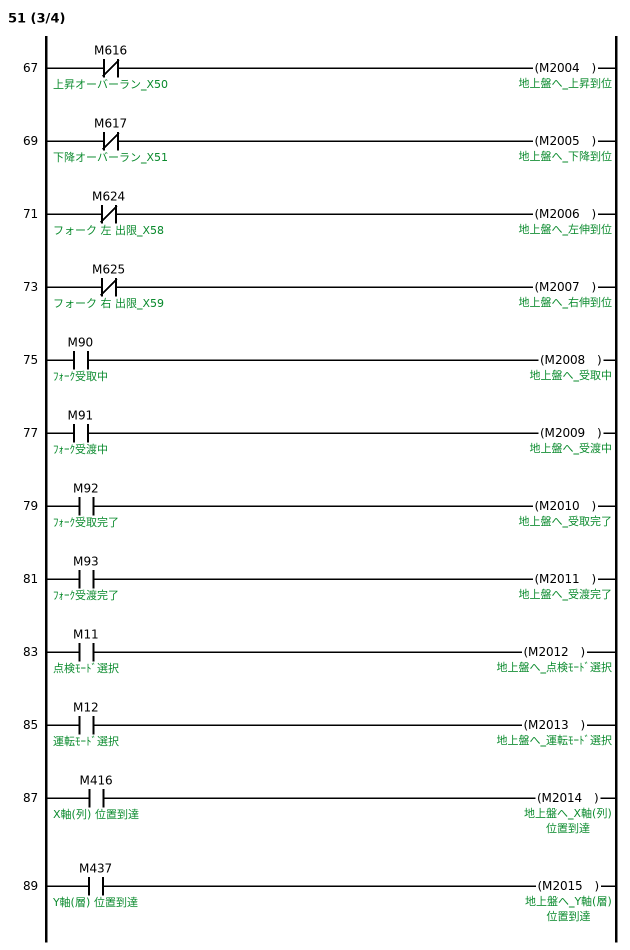
67    LDI     M616  ; 上昇オーバーラン_X50
      OUT     M2004  ; 地上盤へ_上昇到位
69    LDI     M617  ; 下降オーバーラン_X51
      OUT     M2005  ; 地上盤へ_下降到位
71    LDI     M624  ; フォーク 左 出限_X58
      OUT     M2006  ; 地上盤へ_左伸到位
73    LDI     M625  ; フォーク 右 出限_X59
      OUT     M2007  ; 地上盤へ_右伸到位
75    LD      M90  ; ﾌｫｰｸ受取中
      OUT     M2008  ; 地上盤へ_受取中
77    LD      M91  ; ﾌｫｰｸ受渡中
      OUT     M2009  ; 地上盤へ_受渡中
79    LD      M92  ; ﾌｫｰｸ受取完了
      OUT     M2010  ; 地上盤へ_受取完了
81    LD      M93  ; ﾌｫｰｸ受渡完了
      OUT     M2011  ; 地上盤へ_受渡完了
83    LD      M11  ; 点検ﾓｰﾄﾞ選択
      OUT     M2012  ; 地上盤へ_点検ﾓｰﾄﾞ選択
85    LD      M12  ; 運転ﾓｰﾄﾞ選択
      OUT     M2013  ; 地上盤へ_運転ﾓｰﾄﾞ選択
87    LD      M416  ; X軸(列) 位置到達
      OUT     M2014  ; 地上盤へ_X軸(列) 位置到達
89    LD      M437  ; Y軸(層) 位置到達
      OUT     M2015  ; 地上盤へ_Y軸(層) 位置到達
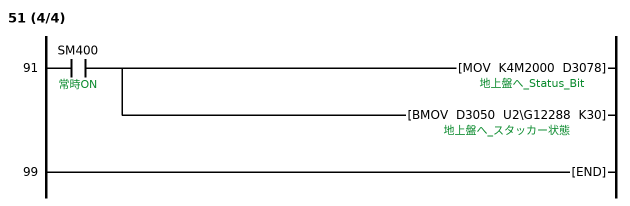
91    LD      SM400  ; 常時ON
      MOV     K4M2000 D3078  ; 地上盤へ_Status_Bit
      BMOV    D3050 U2\G12288 K30
99    END
END_PROGRAM

PROGRAM 52  // Ether 出力 SEW INV
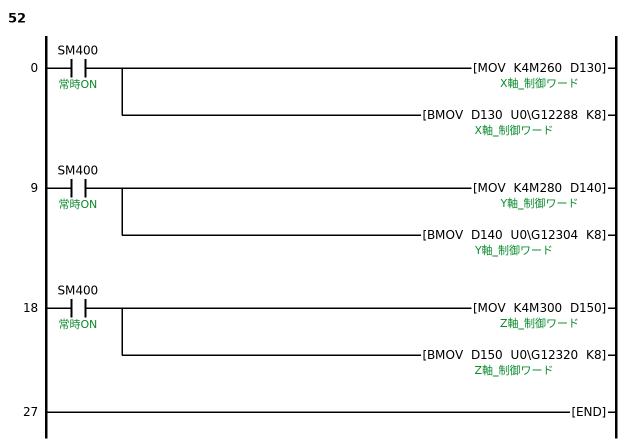
0     LD      SM400  ; 常時ON
      MOV     K4M260 D130  ; X軸_Enable非常停止 / X軸_制御ワード
      BMOV    D130 U0\G12288 K8
9     LD      SM400  ; 常時ON
      MOV     K4M280 D140  ; Y軸_Enable非常停止 / Y軸_制御ワード
      BMOV    D140 U0\G12304 K8
18    LD      SM400  ; 常時ON
      MOV     K4M300 D150  ; Z軸_Enable非常停止 / Z軸_制御ワード
      BMOV    D150 U0\G12320 K8
27    END
END_PROGRAM

PROGRAM 01  // IO入力
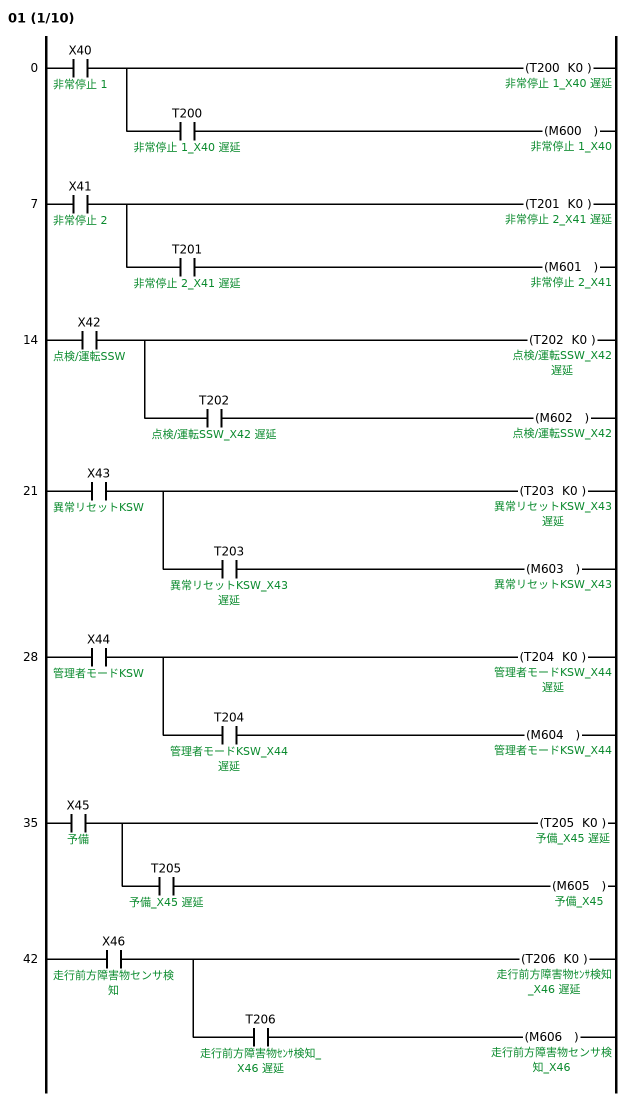
0     LD      X40  ; 非常停止 1
      OUT     T200 K0  ; 非常停止 1_X40 遅延
      AND     T200  ; 非常停止 1_X40 遅延
      OUT     M600  ; 非常停止 1_X40
7     LD      X41  ; 非常停止 2
      OUT     T201 K0  ; 非常停止 2_X41 遅延
      AND     T201  ; 非常停止 2_X41 遅延
      OUT     M601  ; 非常停止 2_X41
14    LD      X42  ; 点検/運転SSW
      OUT     T202 K0  ; 点検/運転SSW_X42 遅延
      AND     T202  ; 点検/運転SSW_X42 遅延
      OUT     M602  ; 点検/運転SSW_X42
21    LD      X43  ; 異常リセットKSW
      OUT     T203 K0  ; 異常リセットKSW_X43 遅延
      AND     T203  ; 異常リセットKSW_X43 遅延
      OUT     M603  ; 異常リセットKSW_X43
28    LD      X44  ; 管理者モードKSW
      OUT     T204 K0  ; 管理者モードKSW_X44 遅延
      AND     T204  ; 管理者モードKSW_X44 遅延
      OUT     M604  ; 管理者モードKSW_X44
35    LD      X45  ; 予備
      OUT     T205 K0  ; 予備_X45 遅延
      AND     T205  ; 予備_X45 遅延
      OUT     M605  ; 予備_X45
42    LD      X46  ; 走行前方障害物センサ検知
      OUT     T206 K0  ; 走行前方障害物ｾﾝｻ検知_X46 遅延
      AND     T206  ; 走行前方障害物ｾﾝｻ検知_X46 遅延
      OUT     M606  ; 走行前方障害物センサ検知_X46
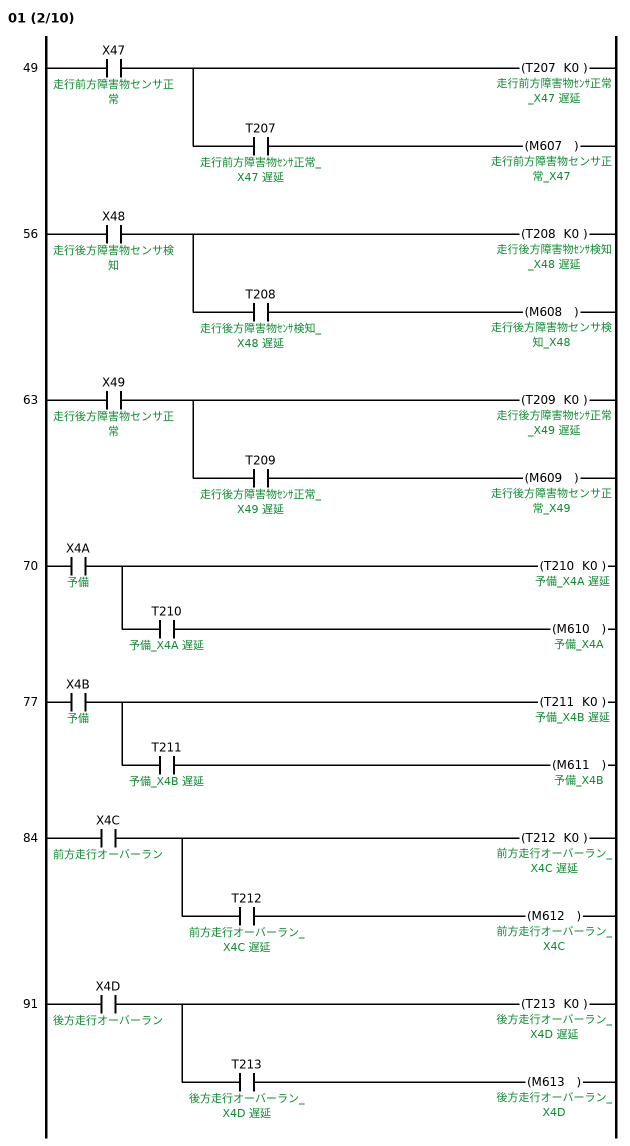
49    LD      X47  ; 走行前方障害物センサ正常
      OUT     T207 K0  ; 走行前方障害物ｾﾝｻ正常_X47 遅延
      AND     T207  ; 走行前方障害物ｾﾝｻ正常_X47 遅延
      OUT     M607  ; 走行前方障害物センサ正常_X47
56    LD      X48  ; 走行後方障害物センサ検知
      OUT     T208 K0  ; 走行後方障害物ｾﾝｻ検知_X48 遅延
      AND     T208  ; 走行後方障害物ｾﾝｻ検知_X48 遅延
      OUT     M608  ; 走行後方障害物センサ検知_X48
63    LD      X49  ; 走行後方障害物センサ正常
      OUT     T209 K0  ; 走行後方障害物ｾﾝｻ正常_X49 遅延
      AND     T209  ; 走行後方障害物ｾﾝｻ正常_X49 遅延
      OUT     M609  ; 走行後方障害物センサ正常_X49
70    LD      X4A  ; 予備
      OUT     T210 K0  ; 予備_X4A 遅延
      AND     T210  ; 予備_X4A 遅延
      OUT     M610  ; 予備_X4A
77    LD      X4B  ; 予備
      OUT     T211 K0  ; 予備_X4B 遅延
      AND     T211  ; 予備_X4B 遅延
      OUT     M611  ; 予備_X4B
84    LD      X4C  ; 前方走行オーバーラン
      OUT     T212 K0  ; 前方走行オーバーラン_X4C 遅延
      AND     T212  ; 前方走行オーバーラン_X4C 遅延
      OUT     M612  ; 前方走行オーバーラン_X4C
91    LD      X4D  ; 後方走行オーバーラン
      OUT     T213 K0  ; 後方走行オーバーラン_X4D 遅延
      AND     T213  ; 後方走行オーバーラン_X4D 遅延
      OUT     M613  ; 後方走行オーバーラン_X4D
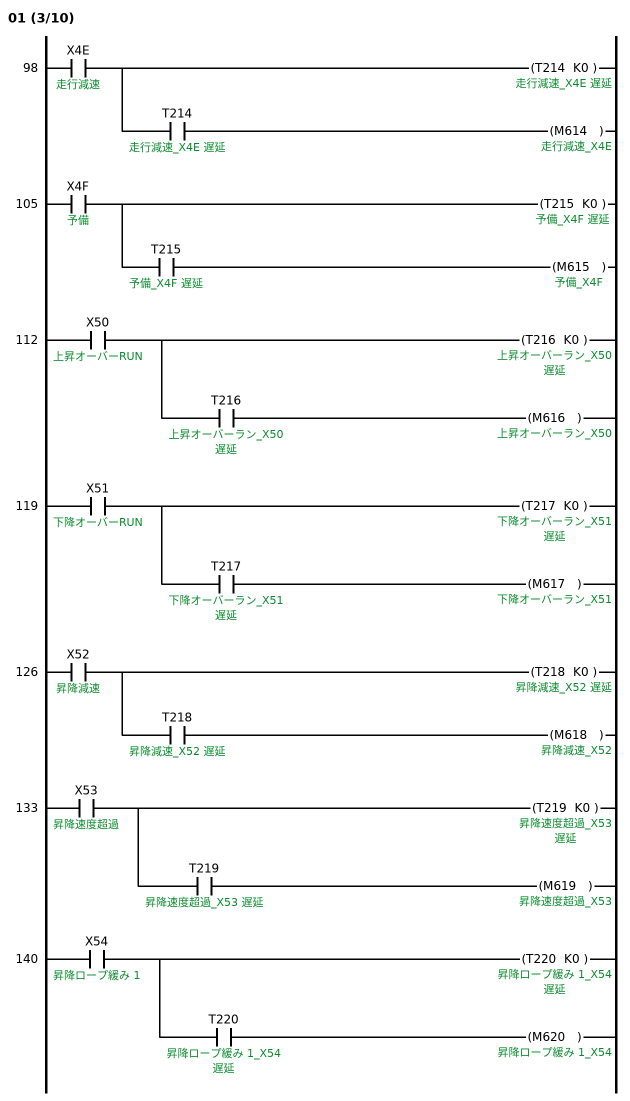
98    LD      X4E  ; 走行減速
      OUT     T214 K0  ; 走行減速_X4E 遅延
      AND     T214  ; 走行減速_X4E 遅延
      OUT     M614  ; 走行減速_X4E
105   LD      X4F  ; 予備
      OUT     T215 K0  ; 予備_X4F 遅延
      AND     T215  ; 予備_X4F 遅延
      OUT     M615  ; 予備_X4F
112   LD      X50  ; 上昇オーバーRUN
      OUT     T216 K0  ; 上昇オーバーラン_X50 遅延
      AND     T216  ; 上昇オーバーラン_X50 遅延
      OUT     M616  ; 上昇オーバーラン_X50
119   LD      X51  ; 下降オーバーRUN
      OUT     T217 K0  ; 下降オーバーラン_X51 遅延
      AND     T217  ; 下降オーバーラン_X51 遅延
      OUT     M617  ; 下降オーバーラン_X51
126   LD      X52  ; 昇降減速
      OUT     T218 K0  ; 昇降減速_X52 遅延
      AND     T218  ; 昇降減速_X52 遅延
      OUT     M618  ; 昇降減速_X52
133   LD      X53  ; 昇降速度超過
      OUT     T219 K0  ; 昇降速度超過_X53 遅延
      AND     T219  ; 昇降速度超過_X53 遅延
      OUT     M619  ; 昇降速度超過_X53
140   LD      X54  ; 昇降ロープ緩み 1
      OUT     T220 K0  ; 昇降ロープ緩み 1_X54 遅延
      AND     T220  ; 昇降ロープ緩み 1_X54 遅延
      OUT     M620  ; 昇降ロープ緩み 1_X54
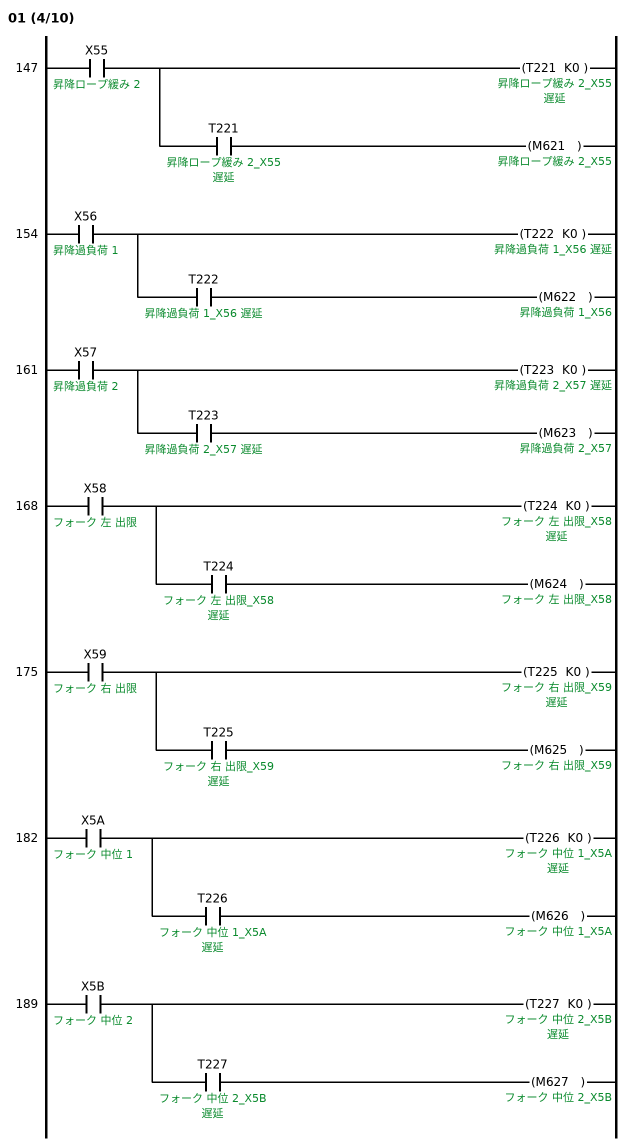
147   LD      X55  ; 昇降ロープ緩み 2
      OUT     T221 K0  ; 昇降ロープ緩み 2_X55 遅延
      AND     T221  ; 昇降ロープ緩み 2_X55 遅延
      OUT     M621  ; 昇降ロープ緩み 2_X55
154   LD      X56  ; 昇降過負荷 1
      OUT     T222 K0  ; 昇降過負荷 1_X56 遅延
      AND     T222  ; 昇降過負荷 1_X56 遅延
      OUT     M622  ; 昇降過負荷 1_X56
161   LD      X57  ; 昇降過負荷 2
      OUT     T223 K0  ; 昇降過負荷 2_X57 遅延
      AND     T223  ; 昇降過負荷 2_X57 遅延
      OUT     M623  ; 昇降過負荷 2_X57
168   LD      X58  ; フォーク 左 出限
      OUT     T224 K0  ; フォーク 左 出限_X58 遅延
      AND     T224  ; フォーク 左 出限_X58 遅延
      OUT     M624  ; フォーク 左 出限_X58
175   LD      X59  ; フォーク 右 出限
      OUT     T225 K0  ; フォーク 右 出限_X59 遅延
      AND     T225  ; フォーク 右 出限_X59 遅延
      OUT     M625  ; フォーク 右 出限_X59
182   LD      X5A  ; フォーク 中位 1
      OUT     T226 K0  ; フォーク 中位 1_X5A 遅延
      AND     T226  ; フォーク 中位 1_X5A 遅延
      OUT     M626  ; フォーク 中位 1_X5A
189   LD      X5B  ; フォーク 中位 2
      OUT     T227 K0  ; フォーク 中位 2_X5B 遅延
      AND     T227  ; フォーク 中位 2_X5B 遅延
      OUT     M627  ; フォーク 中位 2_X5B
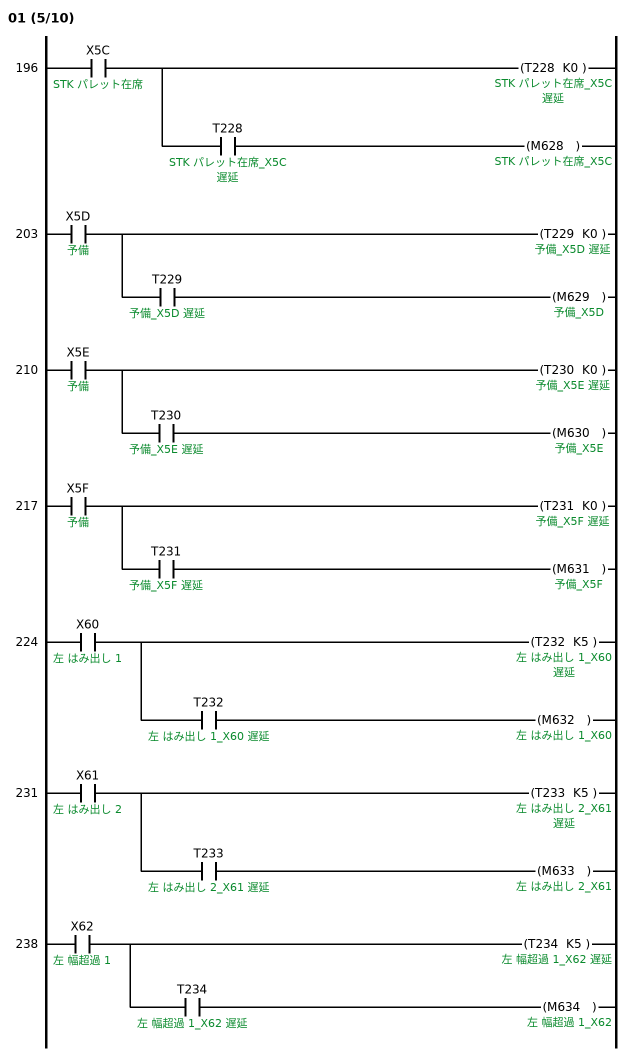
196   LD      X5C  ; STK パレット在席
      OUT     T228 K0  ; STK パレット在席_X5C 遅延
      AND     T228  ; STK パレット在席_X5C 遅延
      OUT     M628  ; STK パレット在席_X5C
203   LD      X5D  ; 予備
      OUT     T229 K0  ; 予備_X5D 遅延
      AND     T229  ; 予備_X5D 遅延
      OUT     M629  ; 予備_X5D
210   LD      X5E  ; 予備
      OUT     T230 K0  ; 予備_X5E 遅延
      AND     T230  ; 予備_X5E 遅延
      OUT     M630  ; 予備_X5E
217   LD      X5F  ; 予備
      OUT     T231 K0  ; 予備_X5F 遅延
      AND     T231  ; 予備_X5F 遅延
      OUT     M631  ; 予備_X5F
224   LD      X60  ; 左 はみ出し 1
      OUT     T232 K5  ; 左 はみ出し 1_X60 遅延
      AND     T232  ; 左 はみ出し 1_X60 遅延
      OUT     M632  ; 左 はみ出し 1_X60
231   LD      X61  ; 左 はみ出し 2
      OUT     T233 K5  ; 左 はみ出し 2_X61 遅延
      AND     T233  ; 左 はみ出し 2_X61 遅延
      OUT     M633  ; 左 はみ出し 2_X61
238   LD      X62  ; 左 幅超過 1
      OUT     T234 K5  ; 左 幅超過 1_X62 遅延
      AND     T234  ; 左 幅超過 1_X62 遅延
      OUT     M634  ; 左 幅超過 1_X62
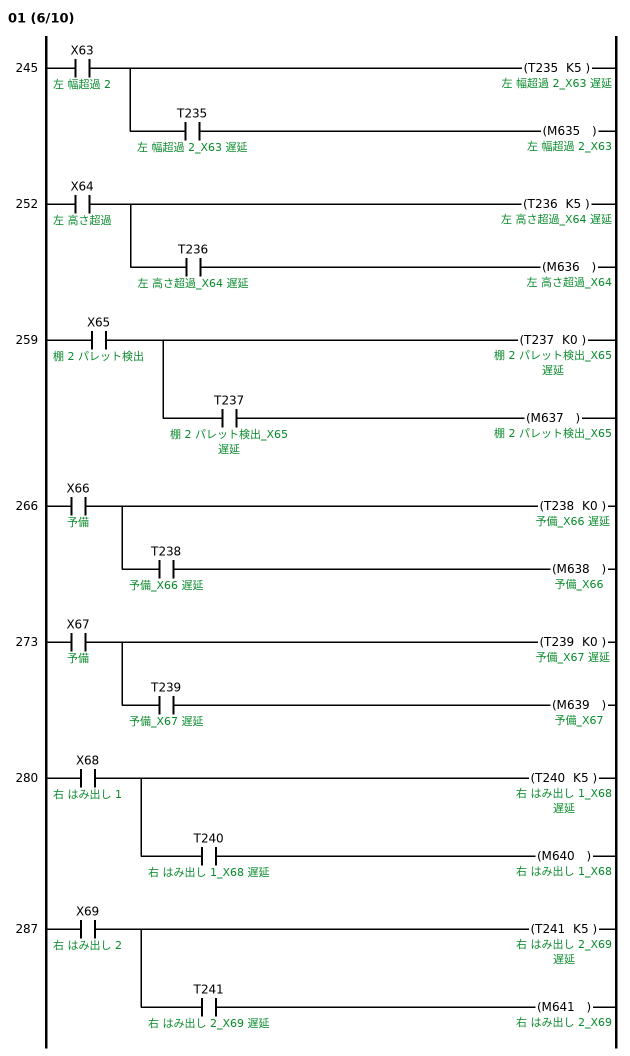
245   LD      X63  ; 左 幅超過 2
      OUT     T235 K5  ; 左 幅超過 2_X63 遅延
      AND     T235  ; 左 幅超過 2_X63 遅延
      OUT     M635  ; 左 幅超過 2_X63
252   LD      X64  ; 左 高さ超過
      OUT     T236 K5  ; 左 高さ超過_X64 遅延
      AND     T236  ; 左 高さ超過_X64 遅延
      OUT     M636  ; 左 高さ超過_X64
259   LD      X65  ; 棚 2 パレット検出
      OUT     T237 K0  ; 棚 2 パレット検出_X65 遅延
      AND     T237  ; 棚 2 パレット検出_X65 遅延
      OUT     M637  ; 棚 2 パレット検出_X65
266   LD      X66  ; 予備
      OUT     T238 K0  ; 予備_X66 遅延
      AND     T238  ; 予備_X66 遅延
      OUT     M638  ; 予備_X66
273   LD      X67  ; 予備
      OUT     T239 K0  ; 予備_X67 遅延
      AND     T239  ; 予備_X67 遅延
      OUT     M639  ; 予備_X67
280   LD      X68  ; 右 はみ出し 1
      OUT     T240 K5  ; 右 はみ出し 1_X68 遅延
      AND     T240  ; 右 はみ出し 1_X68 遅延
      OUT     M640  ; 右 はみ出し 1_X68
287   LD      X69  ; 右 はみ出し 2
      OUT     T241 K5  ; 右 はみ出し 2_X69 遅延
      AND     T241  ; 右 はみ出し 2_X69 遅延
      OUT     M641  ; 右 はみ出し 2_X69
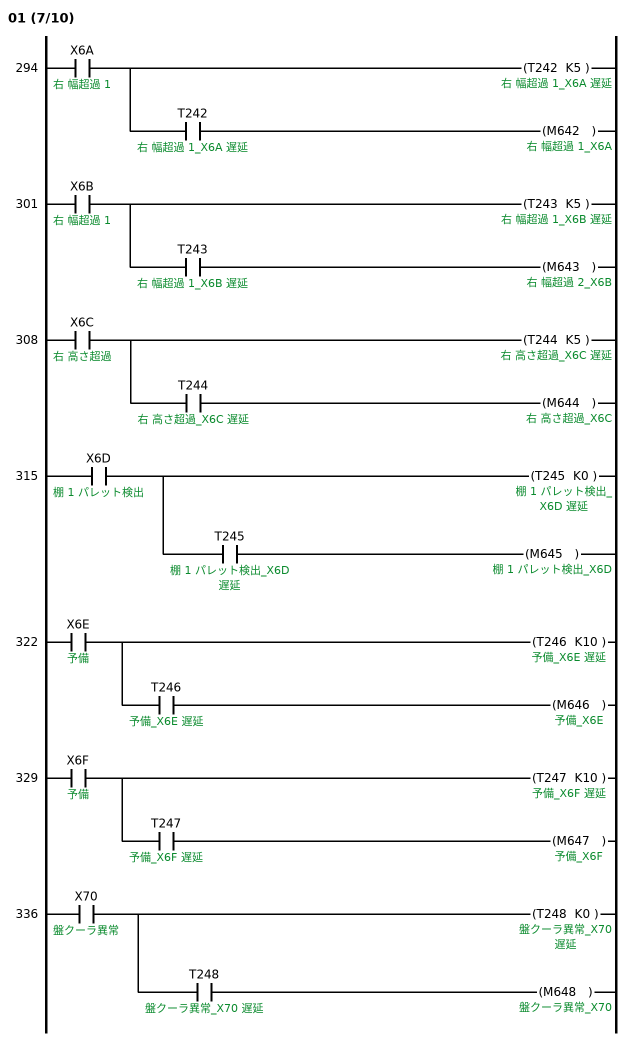
294   LD      X6A  ; 右 幅超過 1
      OUT     T242 K5  ; 右 幅超過 1_X6A 遅延
      AND     T242  ; 右 幅超過 1_X6A 遅延
      OUT     M642  ; 右 幅超過 1_X6A
301   LD      X6B  ; 右 幅超過 1
      OUT     T243 K5  ; 右 幅超過 1_X6B 遅延
      AND     T243  ; 右 幅超過 1_X6B 遅延
      OUT     M643  ; 右 幅超過 2_X6B
308   LD      X6C  ; 右 高さ超過
      OUT     T244 K5  ; 右 高さ超過_X6C 遅延
      AND     T244  ; 右 高さ超過_X6C 遅延
      OUT     M644  ; 右 高さ超過_X6C
315   LD      X6D  ; 棚 1 パレット検出
      OUT     T245 K0  ; 棚 1 パレット検出_X6D 遅延
      AND     T245  ; 棚 1 パレット検出_X6D 遅延
      OUT     M645  ; 棚 1 パレット検出_X6D
322   LD      X6E  ; 予備
      OUT     T246 K10  ; 予備_X6E 遅延
      AND     T246  ; 予備_X6E 遅延
      OUT     M646  ; 予備_X6E
329   LD      X6F  ; 予備
      OUT     T247 K10  ; 予備_X6F 遅延
      AND     T247  ; 予備_X6F 遅延
      OUT     M647  ; 予備_X6F
336   LD      X70  ; 盤クーラ異常
      OUT     T248 K0  ; 盤クーラ異常_X70 遅延
      AND     T248  ; 盤クーラ異常_X70 遅延
      OUT     M648  ; 盤クーラ異常_X70
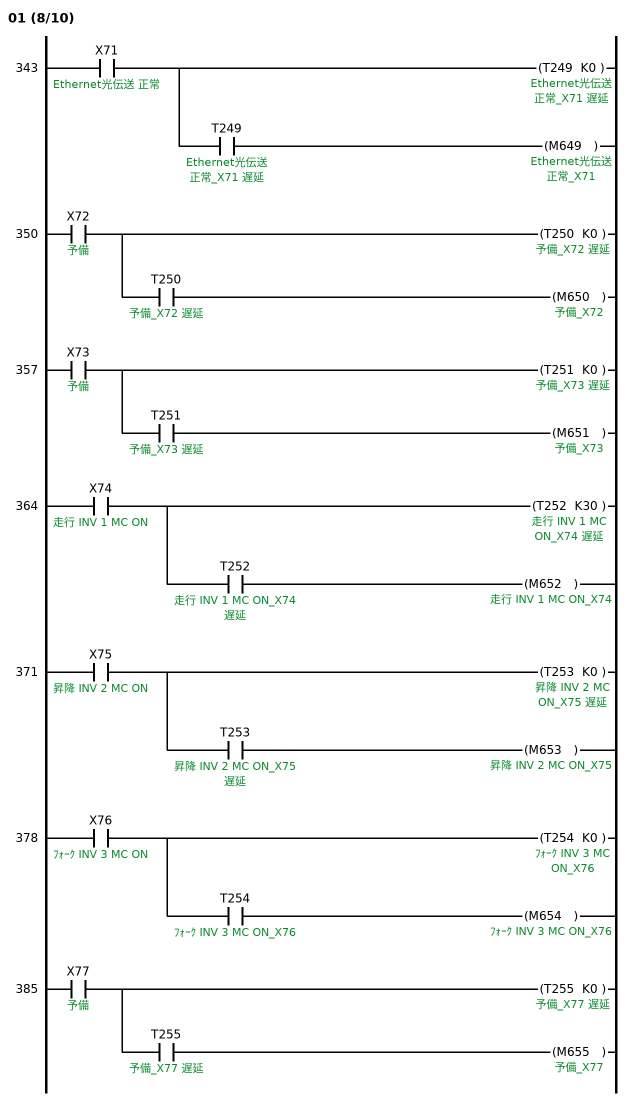
343   LD      X71  ; Ethernet光伝送 正常
      OUT     T249 K0  ; Ethernet光伝送 正常_X71 遅延
      AND     T249  ; Ethernet光伝送 正常_X71 遅延
      OUT     M649  ; Ethernet光伝送 正常_X71
350   LD      X72  ; 予備
      OUT     T250 K0  ; 予備_X72 遅延
      AND     T250  ; 予備_X72 遅延
      OUT     M650  ; 予備_X72
357   LD      X73  ; 予備
      OUT     T251 K0  ; 予備_X73 遅延
      AND     T251  ; 予備_X73 遅延
      OUT     M651  ; 予備_X73
364   LD      X74  ; 走行 INV 1 MC ON
      OUT     T252 K30  ; 走行 INV 1 MC ON_X74 遅延
      AND     T252  ; 走行 INV 1 MC ON_X74 遅延
      OUT     M652  ; 走行 INV 1 MC ON_X74
371   LD      X75  ; 昇降 INV 2 MC ON
      OUT     T253 K0  ; 昇降 INV 2 MC ON_X75 遅延
      AND     T253  ; 昇降 INV 2 MC ON_X75 遅延
      OUT     M653  ; 昇降 INV 2 MC ON_X75
378   LD      X76  ; ﾌｫｰｸ INV 3 MC ON
      OUT     T254 K0  ; ﾌｫｰｸ INV 3 MC ON_X76
      AND     T254  ; ﾌｫｰｸ INV 3 MC ON_X76
      OUT     M654  ; ﾌｫｰｸ INV 3 MC ON_X76
385   LD      X77  ; 予備
      OUT     T255 K0  ; 予備_X77 遅延
      AND     T255  ; 予備_X77 遅延
      OUT     M655  ; 予備_X77
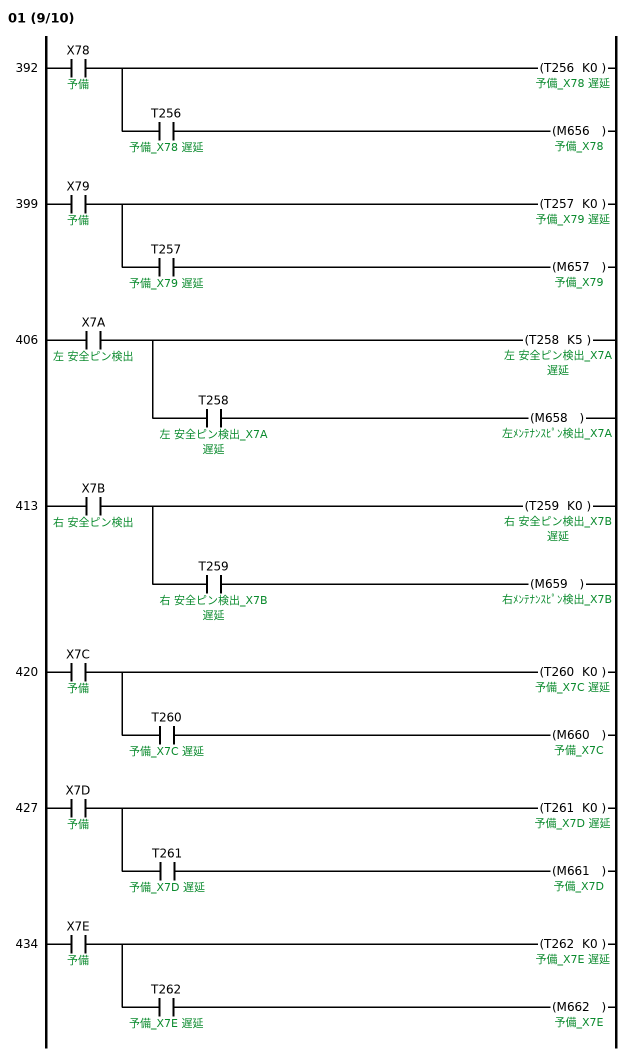
392   LD      X78  ; 予備
      OUT     T256 K0  ; 予備_X78 遅延
      AND     T256  ; 予備_X78 遅延
      OUT     M656  ; 予備_X78
399   LD      X79  ; 予備
      OUT     T257 K0  ; 予備_X79 遅延
      AND     T257  ; 予備_X79 遅延
      OUT     M657  ; 予備_X79
406   LD      X7A  ; 左 安全ピン検出
      OUT     T258 K5  ; 左 安全ピン検出_X7A 遅延
      AND     T258  ; 左 安全ピン検出_X7A 遅延
      OUT     M658  ; 左ﾒﾝﾃﾅﾝｽﾋﾟﾝ検出_X7A
413   LD      X7B  ; 右 安全ピン検出
      OUT     T259 K0  ; 右 安全ピン検出_X7B 遅延
      AND     T259  ; 右 安全ピン検出_X7B 遅延
      OUT     M659  ; 右ﾒﾝﾃﾅﾝｽﾋﾟﾝ検出_X7B
420   LD      X7C  ; 予備
      OUT     T260 K0  ; 予備_X7C 遅延
      AND     T260  ; 予備_X7C 遅延
      OUT     M660  ; 予備_X7C
427   LD      X7D  ; 予備
      OUT     T261 K0  ; 予備_X7D 遅延
      AND     T261  ; 予備_X7D 遅延
      OUT     M661  ; 予備_X7D
434   LD      X7E  ; 予備
      OUT     T262 K0  ; 予備_X7E 遅延
      AND     T262  ; 予備_X7E 遅延
      OUT     M662  ; 予備_X7E
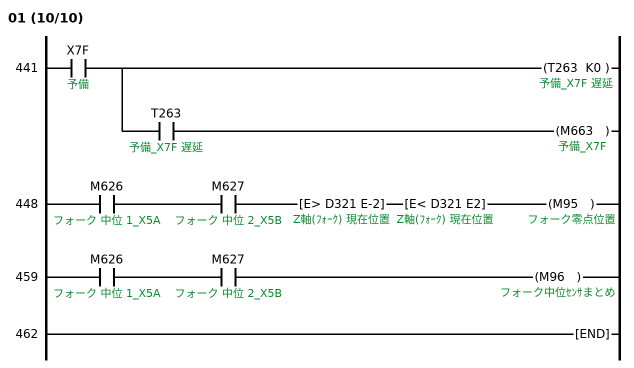
441   LD      X7F  ; 予備
      OUT     T263 K0  ; 予備_X7F 遅延
      AND     T263  ; 予備_X7F 遅延
      OUT     M663  ; 予備_X7F
448   LD      M626  ; フォーク 中位 1_X5A
      AND     M627  ; フォーク 中位 2_X5B
      ANDE>   D321 E-2  ; Z軸(ﾌｫｰｸ) 現在位置
      ANDE<   D321 E2  ; Z軸(ﾌｫｰｸ) 現在位置
      OUT     M95  ; フォーク零点位置
459   LD      M626  ; フォーク 中位 1_X5A
      AND     M627  ; フォーク 中位 2_X5B
      OUT     M96  ; フォーク中位ｾﾝｻまとめ
462   END
END_PROGRAM

// device comments not shown above
D3270  ; ﾌｫｰｸ座標  [1]
M0  ; 電源ON後遅延
M70  ; 待機 補助
M74  ; 受取位置へ 補助
M79  ; 受渡点へ 補助
M147  ; Z軸ON 位置決め_自動_補助 6
M148  ; Z軸ON 位置決め_自動_補助 7
M149  ; Z軸ON 位置決め_自動_補助 8
M201  ; X軸_STO非アクティブ
M202  ; X軸_出力段Enabled
M203  ; X軸_ブレーキオープン済み
M204  ; X軸_モーター回転
M206  ; X軸_新しい相対位置適用済み
M209  ; X軸_ワーニング
M210  ; X軸_ドライブ機構2 有効
M211  ; X軸_メッセージ実速度比較
M212  ; X軸_リミットスイッチ非アク
M213  ; X軸_予備
M214  ; X軸_待機運転有効
M215  ; X軸_HandshakeOut
M221  ; Y軸_STO非アクティブ
M222  ; Y軸_出力段已Enable
M223  ; Y軸_ブレーキオープン済み
M224  ; Y軸_モーター回転
M226  ; Y軸_新しい相対位置適用済み
M229  ; Y軸_ワーニング
M230  ; Y軸_ドライブ機構2 有効
M231  ; Y軸_メッセージ実速度比較
M232  ; Y軸_リミットスイッチ非アク
M233  ; Y軸_予備
M235  ; Y軸_HandshakeOut
M241  ; Z軸_STO非アクティブ
M242  ; Z軸_出力段已Enable
M243  ; Z軸_ブレーキオープン済み
M244  ; Z軸_モーター回転
M246  ; Z軸_新しい相対位置適用済み
M249  ; Z軸_ワーニング
M250  ; Z軸_ドライブ機構2 有効
M251  ; Z軸_メッセージ実速度比較
M252  ; Z軸_リミットスイッチ非アク
M253  ; Z軸_予備
M254  ; Z軸_待機運転有効
M255  ; Z軸_HandshakeOut
M262  ; X軸_予備1
M263  ; X軸_ブレーキ開放
M266  ; X軸_相対位置受信中
M269  ; X軸_予備2
M270  ; X軸_ドライブ機構2 有効
M271  ; X軸_予備3
M272  ; X軸_禁用リミットスイッ
M273  ; X軸_出力段ロック 有効
M274  ; X軸_待機運転有効
M275  ; X軸_HandshakeIn
M282  ; Y軸_予備1
M283  ; Y軸_ブレーキ開放
M286  ; Y軸_相対位置受信中
M289  ; Y軸_予備2
M291  ; Y軸_予備3
M292  ; Y軸_禁用リミットスイッ
M293  ; Y軸_出力段ロック 有効
M295  ; Y軸_HandshakeIn
M302  ; Z軸_予備1
M303  ; Z軸_ブレーキ開放
M306  ; Z軸_相対位置受信中
M309  ; Z軸_予備2
M310  ; Z軸_駆動機構作動
M311  ; Z軸_予備3
M312  ; Z軸_禁用リミットスイッ
M313  ; Z軸_出力段ロック 有効
M314  ; Z軸_待機運転有効
M315  ; Z軸_HandshakeIn
M400  ; X軸ON 位置決め0
M403  ; X軸ON 位置決め3
M404  ; X軸ON 位置決め4
M405  ; X軸ON 位置決め5
M406  ; X軸ON 位置決め6
M407  ; X軸ON 位置決め7
M408  ; X軸ON 位置決め8
M409  ; X軸ON 位置決め9
M410  ; X軸ON 位置決め10
M411  ; X軸ON 位置決め11
M412  ; X軸ON 位置決め12
M413  ; X軸ON 位置決め13
M414  ; X軸ON 位置決め14
M415  ; X軸ON 位置決め15
M421  ; Y軸ON 位置決め0
M424  ; Y軸ON 位置決め3
M425  ; Y軸ON 位置決め4
M426  ; Y軸ON 位置決め5
M427  ; Y軸ON 位置決め6
M428  ; Y軸ON 位置決め7
M429  ; Y軸ON 位置決め8
M430  ; Y軸ON 位置決め9
M431  ; Y軸ON 位置決め10
M432  ; Y軸ON 位置決め11
M433  ; Y軸ON 位置決め12
M434  ; Y軸ON 位置決め13
M435  ; Y軸ON 位置決め14
M436  ; Y軸ON 位置決め15
M442  ; Z軸ON 位置決め0
M445  ; Z軸ON 位置決め3
M446  ; Z軸ON 位置決め4
M447  ; Z軸ON 位置決め5
M448  ; Z軸ON 位置決め6
M449  ; Z軸ON 位置決め7
M450  ; Z軸ON 位置決め8
M451  ; Z軸ON 位置決め9
M452  ; Z軸ON 位置決め10
M453  ; Z軸ON 位置決め11
M454  ; Z軸ON 位置決め12
M455  ; Z軸ON 位置決め13
M456  ; Z軸ON 位置決め14
M457  ; Z軸ON 位置決め15
M921  ; 安全機器一時解除有効
M990  ; テスト用
M2514  ; 地上盤から_予備3
M2515  ; 地上盤から_予備4
M2516  ; 地上盤から_予備5
M2517  ; 地上盤から_予備6
M3196  ; フォーク右側超高アラーム
M3197  ; フォーク右超ワイドアラーム2
M3198  ; フォーク右超ワイドアラーム1
M3199  ; フォーク右側崩壊アラーム2
M3200  ; フォーク右側崩壊アラーム1
M3201  ; フォーク左側超高アラーム
M3202  ; フォーク左超ワイドアラーム2
M3203  ; フォーク左超ワイドアラーム1
M3204  ; フォーク左側崩壊アラーム2
M3205  ; フォーク左側崩壊アラーム1
M3206  ; 搬入可能
M3207  ; 搬出可能
M3230  ; DockTable1搬入可能2
M3231  ; DockTable2搬入可能2
M3232  ; DockTable1搬出可能1
M3233  ; DockTable2搬出可能1
D2  ; GOTｵｰﾊﾞﾗｯﾌﾟｳｨﾝﾄﾞｳ2
D3  ; GOTｵｰﾊﾞﾗｯﾌﾟｳｨﾝﾄﾞｳ3
D4  ; GOTｵｰﾊﾞﾗｯﾌﾟｳｨﾝﾄﾞｳ4
D5  ; GOTｵｰﾊﾞﾗｯﾌﾟｳｨﾝﾄﾞｳ5
D10  ; GOTｼｽﾃﾑ信号1-1
D11  ; GOTｼｽﾃﾑ信号2-1
D12  ; GOT表示中画面番号
D13  ; 表示中ｳｨﾝﾄﾞｳ画面1番号
D14  ; 表示中ｳｨﾝﾄﾞｳ画面2番号
D15  ; 表示中ｳｨﾝﾄﾞｳ画面3番号
D16  ; 表示中ｳｨﾝﾄﾞｳ画面4番号
D17  ; 表示中ｳｨﾝﾄﾞｳ画面5番号
D104  ; X軸(列)_数字入力
D105  ; X軸(列)_現在応用モード
D114  ; Y軸(層)_数字入力
D115  ; Y軸(層)_現在応用モード
D124  ; Z軸(ﾌｫｰｸ)_数字入力
D125  ; Z軸(ﾌｫｰｸ)_現在応用モード
D134  ; X軸_仮想入力端子
D144  ; Y軸_仮想入力端子
D154  ; Z軸_仮想入力端子
D201  ; Auto_列目標位置
D202  ; Auto_列位置決め速度
D203  ; Auto_列位置決め速度
D205  ; X軸(列)_現在位置
D207  ; X軸(列)_現在速度
D209  ; X軸へ_列目標位置
D210  ; Auto_列目標速度
D211  ; Auto_列目標速度
D213  ; Auto_層目標位置
D214  ; Auto_層位置決め速度
D215  ; Auto_層位置決め速度
D217  ; Y軸(層)_現在位置
D219  ; Y軸(層)_現在速度
D221  ; Y軸へ_層目標位置
D222  ; Auto_層目標速度
D223  ; Auto_層目標速度
D225  ; Auto_ﾌｫｰｸ目標位置
D226  ; Auto_ﾌｫｰｸ位置決め速度
D227  ; Auto_ﾌｫｰｸ位置決め速度
D229  ; Z軸(ﾌｫｰｸ)_現在位置
D231  ; Z軸(ﾌｫｰｸ)_現在速度
D233  ; Z軸へ_ﾌｫｰｸ目標位置
D234  ; Auto_ﾌｫｰｸ目標速度
D235  ; Auto_ﾌｫｰｸ目標速度
D302  ; 自動_タスクタイプ
D313  ; 自動_現在タスクID
D315  ; タスク総実行回数
D318  ; X軸(列) 現在位置
D320  ; Y軸(層) 現在位置
D322  ; Z軸(ﾌｫｰｸ) 現在位置
D324  ; X軸(列) 現在速度
D326  ; Y軸(層) 現在速度
D328  ; Z軸(ﾌｫｰｸ) 現在速度
D332  ; オンライン_タスクID
D346  ; 地上→モード
D381  ; X軸位置 決め位置
D383  ; Y軸位置 決め位置
D385  ; Z軸位置 決め位置
D1001  ; X軸(列) モータ現在位置
D1003  ; X軸(列) 位置差
D1005  ; Y軸(層) モータ現在位置
D1007  ; Y軸(層) 位置差
D1009  ; Z軸(ﾌｫｰｸ) モータ現在位置
D1011  ; Z軸(ﾌｫｰｸ) 位置差
D3002  ; 地上盤から_タスクID
D3056  ; 地上盤へ_タスク総実行回数
D3057  ; 地上盤へ_タスク総実行回数
D3253  ; 記録_タスクタイプ
D3255  ; 記録_現在タスクID
D3257  ; 記録_モード
D3261  ; 手動_Z軸位置決め位置Temp
D3263  ; 手動_Y軸位置決め位置Temp
D3265  ; 手動_X軸位置決め位置Temp
D3267  ; ﾊﾟﾚｯﾄ受渡高さ補正値
D3269  ; ﾊﾟﾚｯﾄ受取高さ補正値
D3271  ; ﾌｫｰｸ座標  [1]
D3272  ; ﾌｫｰｸ座標  [2]
D3273  ; ﾌｫｰｸ座標  [2]
D3275  ; 層座標  [1]
D3276  ; 層座標  [2]
D3277  ; 層座標  [2]
D3278  ; 層座標  [3]
D3279  ; 層座標  [3]
D3280  ; 層座標  [4]
D3281  ; 層座標  [4]
D3282  ; 層座標  [5]
D3283  ; 層座標  [5]
D3285  ; 列座標  [1]
D3286  ; 列座標  [2]
D3287  ; 列座標  [2]
D3288  ; 列座標  [3]
D3289  ; 列座標  [3]
D3290  ; 列座標  [4]
D3291  ; 列座標  [4]
D3292  ; 列座標  [5]
D3293  ; 列座標  [5]
D3294  ; 列座標  [6]
D3295  ; 列座標  [6]
D3297  ; 列座標  [7]
D3298  ; 列座標  [8]
D3299  ; 列座標  [8]
D3301  ; 列座標  [9]
D3302  ; 列座標  [10]
D3303  ; 列座標  [10]
D3304  ; 列座標  [11]
D3305  ; 列座標  [11]
D3306  ; 列座標  [12]
D3307  ; 列座標  [12]
D3308  ; 列座標  [13]
D3309  ; 列座標  [13]
D3310  ; 列座標  [14]
D3311  ; 列座標  [14]
D5013  ; ﾊﾟﾗﾒｰﾀ_X軸 前 リミット設置SP
D5015  ; ﾊﾟﾗﾒｰﾀ_X軸 後 リミット設置SP
D5017  ; ﾊﾟﾗﾒｰﾀ_Y軸 上 リミット設置SP
D5019  ; ﾊﾟﾗﾒｰﾀ_Y軸 下 リミット設置SP
D5021  ; ﾊﾟﾗﾒｰﾀ_Z軸 左 リミット設置SP
D5023  ; ﾊﾟﾗﾒｰﾀ_Z軸 右 リミット設置SP
D5025  ; ﾊﾟﾗﾒｰﾀ_X軸位置 オフセット量SP
D5027  ; ﾊﾟﾗﾒｰﾀ_Y軸位置 オフセット量SP
D5029  ; ﾊﾟﾗﾒｰﾀ_Z軸位置 オフセット量SP
D5034  ; 搬入出台座標算出基準  列座標0
D5035  ; 搬入出台座標算出基準  列座標0
D5036  ; 搬入出台座標算出基準  層座標0
D5037  ; 搬入出台座標算出基準  層座標0
D5038  ; 搬入出台座標算出基準  排座標0
D5039  ; 搬入出台座標算出基準  排座標0
D5041  ; ﾊﾟﾗﾒｰﾀ_入庫搬入台  列座標1
D5043  ; ﾊﾟﾗﾒｰﾀ_入庫搬入台  層座標1
D5045  ; ﾊﾟﾗﾒｰﾀ_入庫搬入台  排座標1
D5047  ; ﾊﾟﾗﾒｰﾀ_出庫搬入台  列座標2
D5049  ; ﾊﾟﾗﾒｰﾀ_出庫搬入台  層座標2
D5051  ; ﾊﾟﾗﾒｰﾀ_出庫搬入台  排座標2
D5052  ; ﾊﾟﾗﾒｰﾀ_入庫搬出台  列座標3
D5053  ; ﾊﾟﾗﾒｰﾀ_入庫搬出台  列座標3
D5054  ; ﾊﾟﾗﾒｰﾀ_入庫搬出台  層座標3
D5055  ; ﾊﾟﾗﾒｰﾀ_入庫搬出台  層座標3
D5057  ; ﾊﾟﾗﾒｰﾀ_入庫搬出台  排座標3
D5058  ; ﾊﾟﾗﾒｰﾀ_出庫搬出台  列座標4
D5059  ; ﾊﾟﾗﾒｰﾀ_出庫搬出台  列座標4
D5060  ; ﾊﾟﾗﾒｰﾀ_出庫搬出台  層座標4
D5061  ; ﾊﾟﾗﾒｰﾀ_出庫搬出台  層座標4
D5063  ; ﾊﾟﾗﾒｰﾀ_出庫搬出台  排座標4
